INTERFACE Awaitable EXTENDS Callable, Resettable, Evaluable

METHOD catchIf : Awaitable
VAR_INPUT
	error: BOOL;
	callback: REFERENCE TO AwaitableError;
	message: STRING(255);
END_VAR
END_METHOD

METHOD continueIf : Awaitable
VAR_INPUT
	value: BOOL;
END_VAR
END_METHOD

METHOD evalue : Awaitable
VAR_INPUT
	value: BOOL;
	onTrueCallback: Callback;
	onFalseCallback: REFERENCE TO AwaitableError;
	message: STRING(255);
END_VAR
END_METHOD

METHOD raiseIf : Awaitable
VAR_INPUT
	error: BOOL;
	callback: REFERENCE TO AwaitableError;
	message: STRING(255);
END_VAR
END_METHOD

END_INTERFACE

(* stored: Version 1.1.0.1, ProductVersion 3.1.4024.12
   Itf Awaitable: Id {6ab0156e-171d-4564-b90d-8e010883ecee}
   Method catchIf: Id {1ae9d2b8-9fa4-47e8-aa05-c5a81386204e}
   Method continueIf: Id {31980aa7-791b-4a07-8e4a-b0531a456d11}
   Method evalue: Id {eb343bfe-5422-49b0-86d4-b2b7caa0cbe6}
   Method raiseIf: Id {c2921e7e-af76-4849-b647-f81cd5fec7a0} *)
